FUNCTION_BLOCK Current_Transformer (* Composite Function Block Type *)
  (* Standard: 61499-2 *)
  (* Version 0.0, 12/10/2023, Cheyan, Schneider Electric, template *)
  PACKAGE Main;
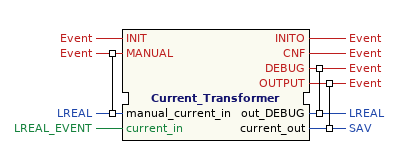
  EVENT_INPUT
    INIT; (* Initialization Request *)
    MANUAL WITH manual_current_in;
  END_EVENT
  EVENT_OUTPUT
    INITO; (* Initialization Confirm *)
    CNF; (* Execution Confirmation *)
    DEBUG WITH out_DEBUG;
    OUTPUT WITH current_out;
  END_EVENT
  VAR_INPUT
    manual_current_in : LREAL;
  END_VAR
  VAR_OUTPUT
    out_DEBUG : LREAL;
    current_out : SAV; (* Output event qualifier *)
  END_VAR
  SOCKETS
    current_in : LREAL_EVENT;
  END_SOCKETS
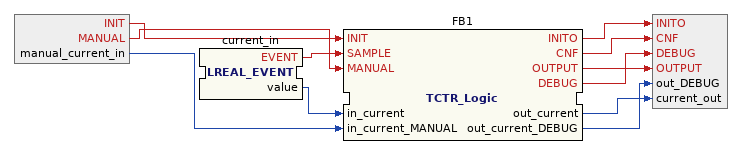
  FBS
    FB1 : TCTR_Logic;
  END_FBS
  EVENT_CONNECTIONS
    INIT TO FB1.INIT;
    FB1.INITO TO INITO;
    FB1.CNF TO CNF;
    current_in.EVENT TO FB1.SAMPLE;
    FB1.DEBUG TO DEBUG;
    MANUAL TO FB1.MANUAL;
    FB1.OUTPUT TO OUTPUT;
  END_CONNECTIONS
  DATA_CONNECTIONS
    current_in.value TO FB1.in_current;
    FB1.out_current_DEBUG TO out_DEBUG;
    manual_current_in TO FB1.in_current_MANUAL;
    FB1.out_current TO current_out;
  END_CONNECTIONS
END_FUNCTION_BLOCK
